// TIA Portal V21 export
DATA_BLOCK "Conteggi"   // DB21
{ S7_Optimized_Access := 'TRUE' }
// stored: MemoryReserve 100
   VAR
      C : Array[0.."K_NumConteggio"] of "Std_Conteggi";
   END_VAR
BEGIN
   // C[0] : Non usare
   C[0].Dati.MemStatoIngConteggio := FALSE;
   C[0].Dati.ActConteggio := 0;
   C[0].Dati.SimulazioneIngresso := FALSE;
END_DATA_BLOCK
